// TIA Portal V19 export
DATA_BLOCK "ItemStatus"   // DB14
{ S7_Optimized_Access := 'TRUE' }
AUTHOR : FLA
FAMILY : UHT
VERSION : 1.0
// stored: AutoNumber false, MemoryReserve 0
   VAR RETAIN
      Y0101 : "ItemStatus_UDT";   // Product inlet valve
      Y0103 : "ItemStatus_UDT";   // Cip / steam inlet valve
      Y0104 : "ItemStatus_UDT";   // Cip / steam inlet valve
      Y0109 : "ItemStatus_UDT";   // Cooling water to jacket valve
      Y0111 : "ItemStatus_UDT";   // Sterile air inlet valve
      Y0112 : "ItemStatus_UDT";   // Filling line stop valve
      Y0113 : "ItemStatus_UDT";   // Filling line steam / cip valve
      Y0114 : "ItemStatus_UDT";   // Cip return / drain valve
      Y0115 : "ItemStatus_UDT";   // Water to balance tank valve
      M0139 : "ItemStatus_UDT";   // Cip pump
      Y0116 : "ItemStatus_UDT";   // Cip return from tank/filling
      Y0108 : "ItemStatus_UDT";   // Steam / cip to valve 01.01
      Y0117 : "ItemStatus_UDT";   // Cip
      Y0118 : "ItemStatus_UDT";   // Steam valve
      Y0237 : "ItemStatus_UDT";   // Relay signal to uht request lye
      Y0238 : "ItemStatus_UDT";   // Relay signal to uht request acid
      Y0119 : "ItemStatus_UDT";   // Flush chain wash
      Y0124 : "ItemStatus_UDT";   // By-pass valve steam valve 01.01
      Y0135_NOT_USED : "ItemStatus_UDT";   // Condensate valve agitator
      Y0136_NOT_USED : "ItemStatus_UDT";   // Steam to condenstate valve
      Y0137_NOT_USED : "ItemStatus_UDT";   // Water to condensater valve
      Y0143 : "ItemStatus_UDT";   // Drain valve bottom sterile filter
      Y0144_NOT_USED : "ItemStatus_UDT";   // Drain valve cip 01.01
      Y0147 : "ItemStatus_UDT";   // Steam valve to 01.13
      Y0148 : "ItemStatus_UDT";   // Steam valve to sterilzing
      Y0158 : "ItemStatus_UDT";   // Steam valve to injector
      Y0545 : "ItemStatus_UDT";   // Steam by-pass valve reduced
      PACK1 : "ItemStatus_UDT";   // Relay signal to packing product availa.
      PACK2 : "ItemStatus_UDT";   // Relay signal to packing product availa.
      PACK3 : "ItemStatus_UDT";   // Relay signal to packing product availa.
      PACK4 : "ItemStatus_UDT";   // Relay signal to packing product availa.
      AlarmLamp : "ItemStatus_UDT";   // Internal alarmlamp
      AHV_CLOSED : "ItemStatus_UDT";   // Ahv barrier closed
      AHV_HIGH_LEVEL : "ItemStatus_UDT";   // Ahv high level
      AHV_READY : "ItemStatus_UDT";   // Ahv ready
      AHV_SHUT_DOWN : "ItemStatus_UDT";   // Ahv shut down
      AHV_STERILE : "ItemStatus_UDT";   // Ahv sterile
      PROD_AVAILABLE : "ItemStatus_UDT";   // Product available
      RINSE_READY : "ItemStatus_UDT";   // Rinse ready
      CAUSTIC_READY : "ItemStatus_UDT";   // Caustic ready
      ACID_READY : "ItemStatus_UDT";   // Acid ready
      CIP_FILLER_ENABLE : "ItemStatus_UDT";   // spare
      WATER_PUMP : "ItemStatus_UDT";   // spare
      Y0901 : "ItemStatus_UDT";   // spare
      Y0902 : "ItemStatus_UDT";   // spare
      Y0903 : "ItemStatus_UDT";   // spare
      TANK_READY : "ItemStatus_UDT";   // Signal to uht tank ready
      TANK_OPEN : "ItemStatus_UDT";   // Signal to uht tank open
      Y0904 : "ItemStatus_UDT";   // spare
      Y0905 : "ItemStatus_UDT";   // spare
      Y0906 : "ItemStatus_UDT";   // spare
      Y0907 : "ItemStatus_UDT";   // spare
      Y0908 : "ItemStatus_UDT";   // spare
      Y0909 : "ItemStatus_UDT";   // spare
      Y0910 : "ItemStatus_UDT";   // spare
      Y0911 : "ItemStatus_UDT";   // spare
      Y0912 : "ItemStatus_UDT";   // spare
      Q41_1 : "ItemStatus_UDT";   // spare
      CIP_Route : "ItemStatus_UDT";   // spare
      SIP_Steam : "ItemStatus_UDT";   // spare
      Product_Available : "ItemStatus_UDT";   // spare
      Barrier_Sterile : "ItemStatus_UDT";   // spare
      Product_Route : "ItemStatus_UDT";   // spare
      X0913 : "ItemStatus_UDT";   // spare
      V0930 : "ItemStatus_UDT";
      V0931 : "ItemStatus_UDT";
      spare2 : "ItemStatus_UDT";
      V0552 : "ItemStatus_UDT";
      V0934 : "ItemStatus_UDT";
      V0935 : "ItemStatus_UDT";
      V0940 : "ItemStatus_UDT";
      V0941 : "ItemStatus_UDT";
      V0942 : "ItemStatus_UDT";
      V0943 : "ItemStatus_UDT";
      V0944 : "ItemStatus_UDT";
      V0945 : "ItemStatus_UDT";
      M0940 : "ItemStatus_UDT";
      V1021 : "ItemStatus_UDT";
      V1023 : "ItemStatus_UDT";
      V1024 : "ItemStatus_UDT";
      V1025 : "ItemStatus_UDT";
      V1027 : "ItemStatus_UDT";
      V1083 : "ItemStatus_UDT";
      M0941 : "ItemStatus_UDT";
      V0936 : "ItemStatus_UDT";
   END_VAR
BEGIN
END_DATA_BLOCK
